Staubli VAL3: libSignals.dtx

bool bSearchLFail
bool bSearchLSuccess
num nBlendOffToll = 0.1
num nBlendOnToll = 0.5
num nMaxTask = 10
num nMovesCount
num nPulseCount
num nSA_Count
num nSE_Count
num nSzoneCount
num nWzoneCount
bool bAdvMoveBusy[20]
string sAdvMovePrefix = "advMove"
bool bAdvMoves
string VERSION = "0.3.2"
num nDeadLockTout = 0.2
